(* PLC project SafeLOGIC-1, BrAutomation SafeDESIGNER  4.2.6.2 *)
(* stored: companyURL http://www.br-automation.com, creationDateTime Mon Sep 25 14:29:29 2023 *)

PROGRAM Main
  VAR  (* added by the conversion: wires and edge detectors of the diagram *)
    _AND_S19_OUT : ANY;
  END_VAR

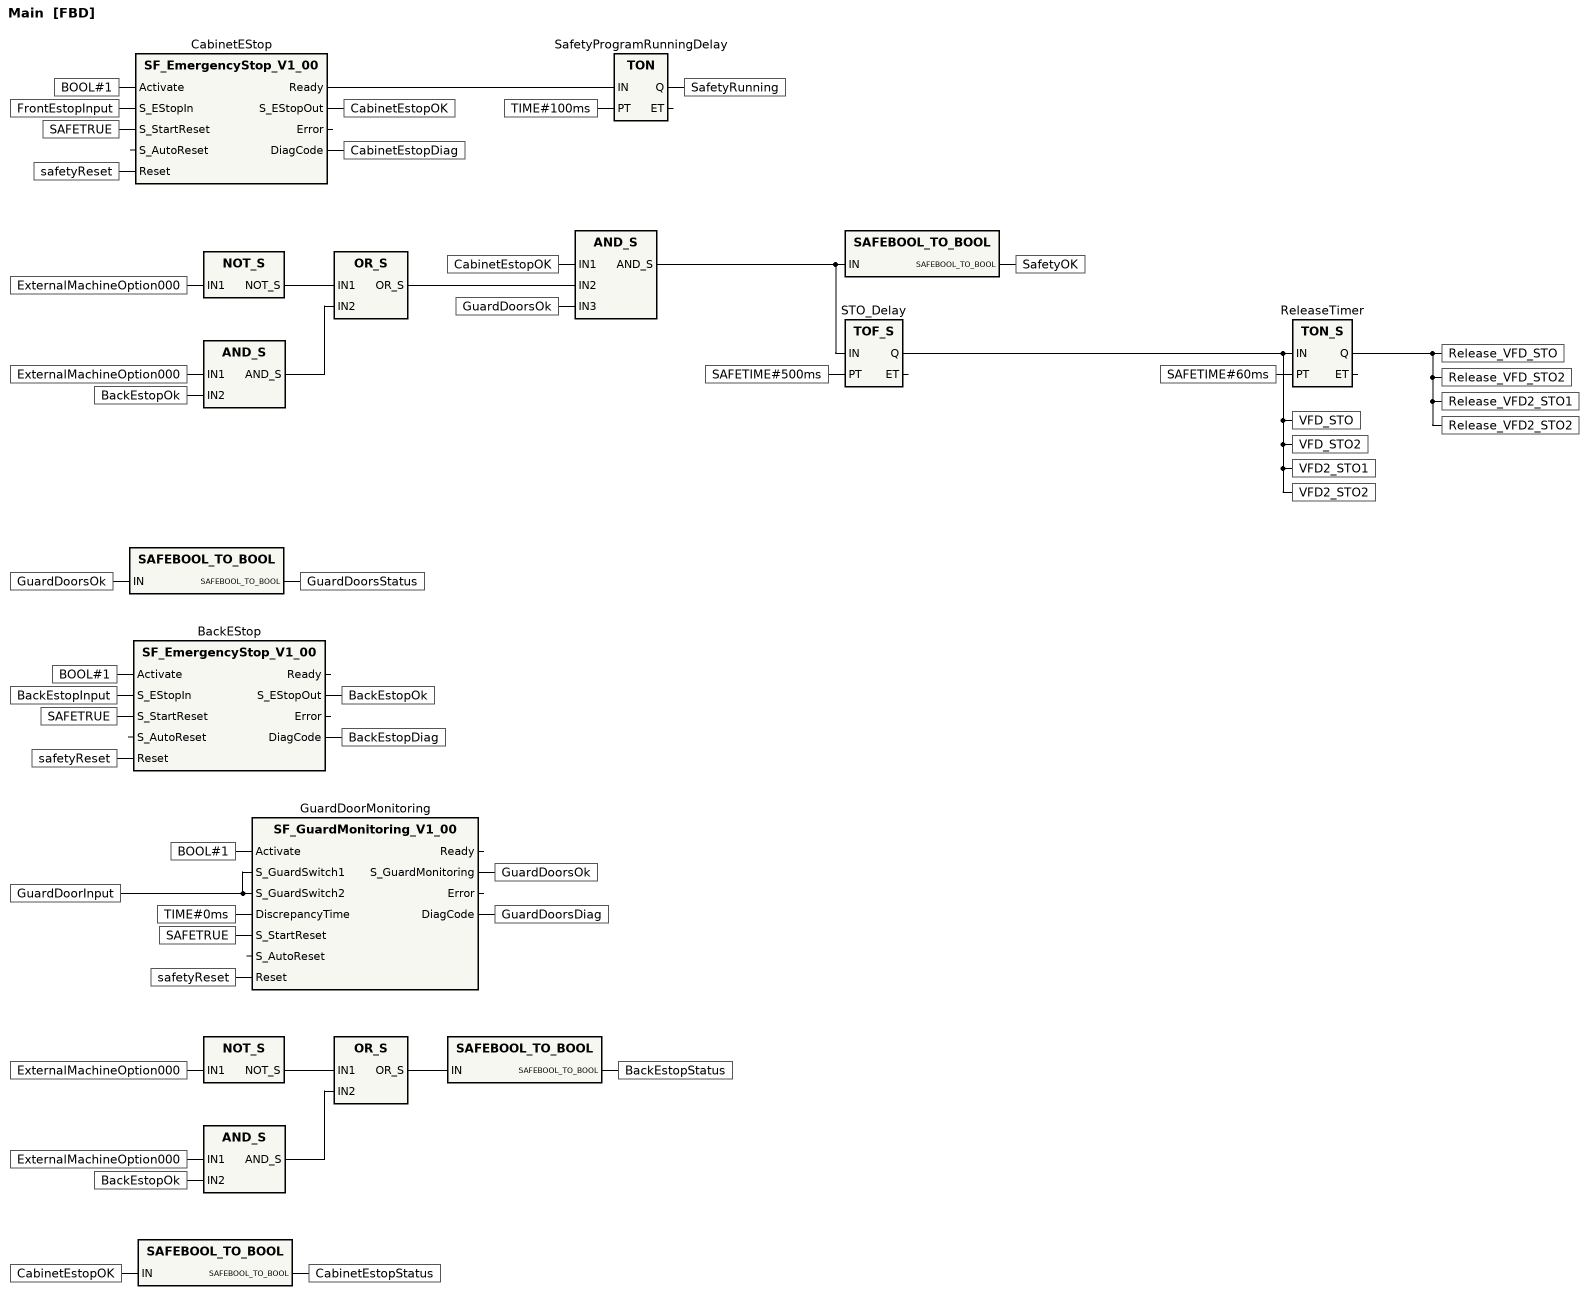
(* FBD diagram, written out as Structured Text *)
CabinetEStop(Activate := BOOL#1, S_EStopIn := FrontEstopInput, S_StartReset := SAFETRUE, Reset := safetyReset);
CabinetEstopDiag := CabinetEStop.DiagCode;
CabinetEstopOK := CabinetEStop.S_EStopOut;
SafetyProgramRunningDelay(IN := CabinetEStop.Ready, PT := TIME#100ms);
SafetyRunning := SafetyProgramRunningDelay.Q;
BackEStop(Activate := BOOL#1, S_EStopIn := BackEstopInput, S_StartReset := SAFETRUE, Reset := safetyReset);
BackEstopOk := BackEStop.S_EStopOut;
BackEstopDiag := BackEStop.DiagCode;
GuardDoorMonitoring(Activate := BOOL#1, S_GuardSwitch1 := GuardDoorInput, S_GuardSwitch2 := GuardDoorInput, DiscrepancyTime := TIME#0ms, S_StartReset := SAFETRUE, Reset := safetyReset);
GuardDoorsDiag := GuardDoorMonitoring.DiagCode;
GuardDoorsOk := GuardDoorMonitoring.S_GuardMonitoring;
_AND_S19_OUT := AND_S(CabinetEstopOK, OR_S(NOT_S(ExternalMachineOption000), AND_S(ExternalMachineOption000, BackEstopOk)), GuardDoorsOk);
STO_Delay(IN := _AND_S19_OUT, PT := SAFETIME#500ms);
VFD_STO := STO_Delay.Q;
SafetyOK := SAFEBOOL_TO_BOOL(_AND_S19_OUT);
VFD_STO2 := STO_Delay.Q;
VFD2_STO1 := STO_Delay.Q;
VFD2_STO2 := STO_Delay.Q;
ReleaseTimer(IN := STO_Delay.Q, PT := SAFETIME#60ms);
Release_VFD2_STO1 := ReleaseTimer.Q;
Release_VFD_STO := ReleaseTimer.Q;
Release_VFD_STO2 := ReleaseTimer.Q;
Release_VFD2_STO2 := ReleaseTimer.Q;
GuardDoorsStatus := SAFEBOOL_TO_BOOL(GuardDoorsOk);
BackEstopStatus := SAFEBOOL_TO_BOOL(OR_S(NOT_S(ExternalMachineOption000), AND_S(ExternalMachineOption000, BackEstopOk)));
CabinetEstopStatus := SAFEBOOL_TO_BOOL(CabinetEstopOK);
END_PROGRAM
